PROGRAM POU_3
VAR
	count:WORD;
	prePushed:BOOL;
	pre: INT;
	fbCal:FBAdd;
	result:WORD;
	x:WORD;
	y:WORD;
	z:word;
END_VAR


IF Variables.Button THEN 
	IF NOT prePushed THEN
		count:=count+1;
		prePushed:=TRUE;
		Variables.LED:=NOT Variables.LED;
	END_IF
ELSE
	prePushed:=FALSE;	
END_IF
	
fbCal(a:=5,b:=3,c=>result);


x:=4;
y:=7;
//count:=Func(1,4);
z:=Func(x,y);

ACTION ACT:

END_ACTION

METHOD PUBLIC METH : BOOL
VAR_INPUT
END_VAR
END_METHOD

METHOD PUBLIC METH_1 : BOOL
VAR_INPUT
END_VAR
END_METHOD

END_PROGRAM

(* stored: Version 1.1.0.1, ProductVersion 3.1.4024.12
   POU POU_3: Id {e9fb6442-46c8-4e88-a00e-ab06a86e777a}, SpecialFunc None
   Action ACT: Id {9012192d-863e-4259-aa25-15a8861058de}
   Method METH: Id {358ada81-a0da-45eb-b466-d33d35766cb8}
   Method METH_1: Id {d93de430-ef48-4e3b-a3d0-e29d17b6d2dc} *)
